// TIA Portal V16 export
// export: Created 2024-04-23T10:19:31.9979432Z, ExportSetting WithDefaults, DisplayName Totally Integrated Automation Portal, DisplayVersion V16 Update 5, DisplayName TIA Portal Version Control Interface, DisplayVersion V16 Update 2, DisplayName TIA Portal Openness, DisplayVersion V16 Update 5, DisplayName TIA Portal Teamcenter Gateway, DisplayVersion V16, DisplayName SINAMICS Startdrive Advanced, DisplayVersion V16, DisplayName SINAMICS Startdrive G130, G150, S120, S150, SINAMICS MV, S210, DisplayVersion V16, DisplayName SINAMICS Startdrive G110M, G120, G120C, G120D, G120P, DisplayVersion V16, DisplayName STEP 7 Professional, DisplayVersion V16 Update 5, DisplayName STEP 7 Safety, DisplayVersion V16, DisplayName WinCC UA Professional, DisplayVersion V16 Update 5
ORGANIZATION_BLOCK "Cyclic interrupt"   // OB30, LAD, CyclicInterrupt
{ S7_Optimized_Access := 'TRUE' }
VERSION : 0.1
// stored: AutoNumber true, IsIECCheckEnabled false, SetENOAutomatically false
   VAR_INPUT
      Initial_Call : Bool;   // Initial call of this OB
      Event_Count : Int;   // Events discarded
   END_VAR
BEGIN

REGION Network 1
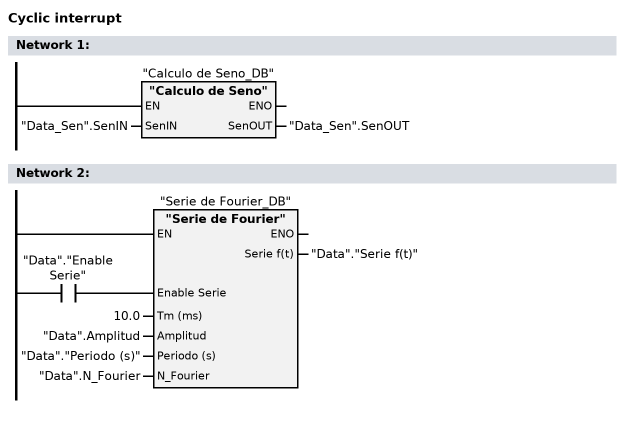
   RUNG wire#powerrail
      "Calculo de Seno_DB"(SenIN := "Data_Sen".SenIN, SenOUT => "Data_Sen".SenOUT)
   END_RUNG
   // the same network as SCL:
   "Calculo de Seno_DB"(SenIN := "Data_Sen".SenIN, SenOUT => "Data_Sen".SenOUT);   // "Calculo de Seno"
END_REGION

REGION Network 2
   RUNG wire#powerrail
      "Serie de Fourier_DB"("Enable Serie" := wire#w1, "Tm (ms)" := 10.0, Amplitud := "Data".Amplitud, "Periodo (s)" := "Data"."Periodo (s)", N_Fourier := "Data".N_Fourier, "Serie f(t)" => "Data"."Serie f(t)")
   END_RUNG
   RUNG wire#powerrail
      Contact( "Data"."Enable Serie" )
   END_RUNG wire#w1
   // the same network as SCL:
   "Serie de Fourier_DB"("Enable Serie" := "Data"."Enable Serie",   // "Serie de Fourier"
                         "Tm (ms)" := 10.0,
                         Amplitud := "Data".Amplitud,
                         "Periodo (s)" := "Data"."Periodo (s)",
                         N_Fourier := "Data".N_Fourier,
                         "Serie f(t)" => "Data"."Serie f(t)");
END_REGION
END_ORGANIZATION_BLOCK
